KUKA KRL program: hp007.src, hp007.dat

--- hp007.src ---
&ACCESS RVP
&REL 111
&COMMENT Princ Accelo Nacional
&PARAM TEMPLATE = C:\KRC\ROBOTER\TEMPLATE\VG_HP
&PARAM EDITMASK = *
DEF hp007( )
;FOLD INI
   ;FOLD BASISTECH INI
      GLOBAL INTERRUPT DECL 3 WHEN $STOPMESS==TRUE DO IR_STOPM ( )
      INTERRUPT ON 3
      BAS (#INITMOV,0 )
   ;ENDFOLD (BASISTECH INI)
   ;FOLD SPOTTECH INI
      USERSPOT(#INIT)
   ;ENDFOLD (SPOTTECH INI)
   ;FOLD GRIPPERTECH INI
      USER_GRP(0,DUMMY,DUMMY,GDEFAULT)
   ;ENDFOLD (GRIPPERTECH INI)
   ;FOLD USER INI
      ;Make your modifications here
         ;FOLD COLLISION_V_3.01 INI
            IF (COLLISION_DATA[1].I_NR>0) THEN
               GLOBAL INTERRUPT DECL 21 WHEN $IN[COLLISION_DATA[1].I_NR]==FALSE DO COLLSTOP (1,0 )
               ENDIF
            IF (COLLISION_DATA[2].I_NR>0) THEN
               GLOBAL INTERRUPT DECL 22 WHEN $IN[COLLISION_DATA[2].I_NR]==FALSE DO COLLSTOP (2,0 )
               ENDIF
            IF (COLLISION_DATA[3].I_NR>0) THEN
               GLOBAL INTERRUPT DECL 23 WHEN $IN[COLLISION_DATA[3].I_NR]==FALSE DO COLLSTOP (3,0 )
               ENDIF
            IF (COLLISION_DATA[4].I_NR>0) THEN
               GLOBAL INTERRUPT DECL 24 WHEN $IN[COLLISION_DATA[4].I_NR]==FALSE DO COLLSTOP (4,0 )
               ENDIF
         ;ENDFOLD (COLLISION_V_3.01 INI)

   ;ENDFOLD (USER INI)
;ENDFOLD (INI)

; Estacao P13.060 - Robo R2
; Programa: Accelo Nacional
; Caracterização dos meios de produção:
; 02/09/2014 09:15 Changes by KUKA Roboter do Brasil

$TIMER[5]=0
$TIMER_STOP[5]=FALSE

chk_w8_wechs_ok ( )  ; CHECK FERRAMENTA: TOOL CHANGE

MBINI( )             ; RESET DOS BITS PARA INICIO DO TRABALHO

  ;FOLD PTP HOME  Vel= 100 % DEFAULT;%{PE}%V2.2.2,%MKUKATPBASIS,%CMOVE,%VPTP,%P 1:PTP, 2:HOME, 3:, 5:100, 7:DEFAULT
  $H_POS=XHOME
  PDAT_ACT=PDEFAULT
  BAS (#PTP_DAT )
  FDAT_ACT=FHOME
  BAS (#FRAMES )
  BAS (#VEL_PTP,100 )
  PTP  XHOME
  ;ENDFOLD

wkz4_an ( )           ; BUSCA PINÇA C3

ps_602c3 ( )          ; SOLDA RESPOT GEO 01

wkz4_ab ( )           ; ENTREGA PINÇA C3

lib_busca_gripper( )  ; LIBERAÇÃO PARA BUSCAR GRIPPER

WKZ2_AN ( )           ; BUSCA GRIPPER ACCELO

ho_st_accelo ( )      ; BUSCA LATEAL NO MAGAZINE

ab_st_accelo ( )      ; DEPOSITA LATERAL GEOBOX

WKZ1_AN ( )           ; BUSCA PINÇA C1

ps_602c1 ( )          ; SOLDA GEOMETRIA E RESPOT C1

end_weld_geometria( ) ; SOLDA GEOMETRIA CONCLUIDA

end_weld_respot ( )   ; SSOLDA RESPOT CONCLUIDA

WKZ1_AB ( )           ; ENTREGA PINÇA C1

WKZ2_off_st_geo ( )   ; BUSCA GRIPPER NA GEOBOX

trabalho_concluido( ) ; TRABALHO CONCLUIDO

WKZ2_AB ( )           ; ENTREGA GRIPPER ACCELO

;FOLD PTP HOME  Vel= 100 % DEFAULT;%{PE}%R 4.1.16,%MKUKATPBASIS,%CMOVE,%VPTP,%P 1:PTP, 2:HOME, 3:, 5:100, 7:DEFAULT
$BWDSTART = FALSE
PDAT_ACT=PDEFAULT
BAS(#PTP_DAT)
FDAT_ACT=FHOME
BAS(#FRAMES)
BAS(#VEL_PTP,100)
$H_POS=XHOME
PTP XHOME
;ENDFOLD

$TIMER_STOP[6]=TRUE

END

--- hp007.dat ---
&ACCESS RVP
&REL 111
&COMMENT Princ Accelo Nacional
&PARAM TEMPLATE = C:\KRC\ROBOTER\TEMPLATE\VG_HP
&PARAM EDITMASK = *
DEFDAT hp007
;FOLD EXTERNAL DECLARATIONS;%{PE}%MKUKATPBASIS,%CEXT,%VCOMMON,%P
   ;FOLD GRIPPERTECH EXT
      EXT  H50 (INT  :IN,INT  :IN,INT  :IN,GRP_TYP  :IN )
   ;ENDFOLD (GRIPPERTECH EXT)
   ;FOLD SPOTTECH EXT
      EXT  USERSPOT (S_COMMAND  :IN,SPOT_TYPE  :IN )
   ;ENDFOLD (SPOTTECH EXT)
   ;FOLD BASISTECH EXT;%{PE}%MKUKATPBASIS,%CEXT,%VEXT,%P
      EXT  BAS (BAS_COMMAND  :IN,REAL  :IN )
      DECL INT SUCCESS
   ;ENDFOLD (BASISTECH EXT)
   ;FOLD USER EXT;%{E}%MKUKATPUSER,%CEXT,%VEXT,%P
      ;Make your modifications here

   ;ENDFOLD (USER EXT)
;ENDFOLD (EXTERNAL DECLARATIONS)

;# ============ START PATH : hp_p13060r2_ltc =============
DECL BASIS_SUGG_T LAST_BASIS={POINT1[] "P1                      ",POINT2[] "P1                      ",CP_PARAMS[] "CPDAT0                  ",PTP_PARAMS[] "PDAT1                   ",CONT[] "                        ",CP_VEL[] "2.0                     ",PTP_VEL[] "100                     "}
ENDDAT
